FUNCTION_BLOCK FB_VRC_NO_FFO_VLS EXTENDS FB_VRC_NO
VAR_IN_OUT
    io_fbFFHWO    :    FB_HardwareFFOutput;
    fbArbiter: FB_Arbiter();
END_VAR
VAR_INPUT
    i_xPMPS_OK:	BOOL	; (*Set to True To switch off the bptm and PMPS Arbiter*)
    i_xIsAperture:BOOL :=FALSE; // Set tp True if this is an Aperture Valve, the MPS Fault will trip only when moving.
    i_sDevName : T_MaxString :=  'VGC'; // Device name for diagnostic
    i_nTransitionRootID: UDINT; //A unique transition Root ID that is equal to or greater than 1000i_xIsAperture:BOOL :=FALSE; // Set tp True if this is an Aperture Valve, the MPS Fault will trip only when moving.
END_VAR
VAR_OUTPUT

END_VAR
VAR

    xPMPS_OK:	BOOL	; (*PMPS interlock*)
    bMoving : BOOL;
    bDone :BOOL;
    tBPTMtimeout:TON;
    bptm: BeamParameterTransitionManager;
    FFO    :    FB_FastFault :=(
        i_DevName := 'VGC',
        i_Desc := 'Fault occurs when the valve is not in safe state',
        i_TypeCode := 16#1010);
    xMPS_OK:	BOOL; (*MPS Fast OK, is set when the Valve is Open*)

END_VAR

(*IO Mapping*)
ACT_IO();

(* On first PLC pass, put valve into vented state, which implies a closed valve *)
IF xFirstPass THEN
    iq_stValve.eVGC_State := Vented;
    iq_stValve.pv_xCLS_SW := FALSE;
    FFO.i_DevName := i_sDevName;
//	iq_stValve.sDevName := i_sDevName;
END_IF


///Check valve position
IF iq_stValve.i_xClsLS AND  iq_stValve.i_xOpnLS THEN
    iq_stValve.eState:=INVALID;
ELSIF NOT iq_stValve.i_xOpnLS AND iq_stValve.i_xClsLS AND iq_stValve. THEN
    iq_stValve.eState:=CLOSED;
ELSIF NOT iq_stValve.i_xClsLS AND iq_stValve.i_xOpnLS AND NOT iq_stValve.q_xOPN_DO THEN
    iq_stValve.eState:=OPEN_F;
ELSIF iq_stValve.i_xClsLS AND NOT iq_stValve.i_xOpnLS AND NOT iq_stValve.q_xOPN_DO THEN
    iq_stValve.eState:=CLOSED;
ELSIF NOT iq_stValve.i_xClsLS AND NOT iq_stValve.i_xOpnLS THEN
    iq_stValve.eState:=MOVING;
ELSE
    iq_stValve.eState:=INVALID;
END_IF




(*PMPS*)
IF NOT(i_xPMPS_OK) THEN
    ACT_PMPS();
END_IF
(*when interlock is lost the Valve closes regardless of the status of the PMPS and EPS*)
xPMPS_OK := i_xPMPS_OK OR (bptm.q_xTransitionAuthorized OR tBPTMtimeout.Q);
IF NOT (iq_stValve.xOPN_OK) THEN
    iq_stValve.pv_xOPN_SW:= FALSE; // Reset switch after inlk is lost
    iq_stValve.q_xOPN_DO := (iq_stValve.pv_xOPN_SW  AND iq_stValve.xOPN_OK) OR (tonOvrd.Q AND i_xOverrideMode);
ELSIF xPMPS_OK THEN
    iq_stValve.q_xOPN_DO := (iq_stValve.pv_xOPN_SW  AND iq_stValve.xOPN_OK) OR (tonOvrd.Q AND i_xOverrideMode);
//ELSIF NOT (i_xPMPS_OK) THEN
    // Only override mode
    //iq_stValve.q_xOPN_DO := (tonOvrd.Q AND i_xOverrideMode);
END_IF

(*MPS Fault setting*)
If (i_xIsAperture ) THEN
    (* When the valve  is open or in Closed position MPS is OK, Fault while moving*)
    xMPS_OK := (i_xOpnLS  AND NOT q_xCLS_DO) XOR (i_xClsLS  AND q_xCLS_DO);
ELSE
    (* When the valve  is open MPS is OK*)
    xMPS_OK := i_xOpnLS AND NOT i_xClsLS AND q_xCLS_DO;
END_IF

(*FAST FAULT*)
FFO(i_xOK := xMPS_OK,
    i_xReset := ,
    i_xAutoReset :=TRUE,
    io_fbFFHWO := io_fbFFHWO);

ACTION ACT_IO:
(*inputs*)
iq_stValve.i_xOpnLS := 	i_xOpnLS;
iq_stValve.i_xClsLS:=	i_xClsLS;
//iq_stValve. := i_xEXT_OK;
iq_stValve.xOverrideMode := i_xOverrideMode;
(*outputs*)
//q_xOPN_DO:= iq_stValve.q_xOPN_DO;
END_ACTION

ACTION ACT_PMPS:
bMoving := (iq_stValve.pv_xOPN_SW AND iq_stValve.i_xClsLS) XOR (NOT iq_stValve.pv_xOPN_SW AND i_xOpnLS);
bDone := (iq_stValve.pv_xOPN_SW AND iq_stValve.i_xOpnLS) XOR (NOT iq_stValve.pv_xOPN_SW AND i_xClsLS);
If (i_xIsAperture ) OR (iq_stValve.pv_xOPN_SW )THEN
    bptm.i_stRequestedAssertion := PMPS_GVL.cstFullBeam;
ELSE  bptm.i_stRequestedAssertion := PMPS_GVL.cst0RateBeam;
END_IF
bptm(fbArbiter:=fbArbiter,
     i_TransitionAssertionID:=i_nTransitionRootID+2,
     i_stTransitionAssertion:=PMPS_GVL.cst0RateBeam,
     i_nRequestedAssertionID:=i_nTransitionRootID+ BOOL_TO_UDINT( iq_stValve.pv_xOPN_SW),
     i_stRequestedAssertion:=,
     i_xMoving:=bMoving,
     i_xDoneMoving:= bDone,
     stCurrentBeamParameters:=PMPS_GVL.stCurrentBeamParameters,
     q_xTransitionAuthorized=>);
// Timeout
tBPTMtimeout(IN:= bMoving AND NOT bptm.q_xTransitionAuthorized , PT:=T#1S);
//xPMPS_OK := bptm.q_xTransitionAuthorized OR tBPTMtimeout.Q;

//Timeout and clear request
IF (tBPTMtimeout.Q) THEN
    fbArbiter.RemoveRequest(bptm.i_TransitionAssertionID);
    fbArbiter.RemoveRequest(bptm.i_nRequestedAssertionID);
END_IF
END_ACTION

METHOD PUBLIC M_IsClosed : BOOL
VAR_INPUT
END_VAR
M_IsClosed := (This^.iq_stValve.eState = E_ValvePositionState.CLOSED);
END_METHOD

METHOD PUBLIC M_IsOpen : BOOL
VAR_INPUT
END_VAR
M_IsOpen := (This^.iq_stValve.eState = E_ValvePositionState.OPEN);
END_METHOD

// Use this Methode to Open or close the valve by setting the OPN_SW to the input value.
METHOD PUBLIC M_Set_CLS_SW : BOOL
VAR_INPUT
        value:BOOL;
END_VAR
This^.iq_stValve.pv_xCLS_SW := value;
END_METHOD

END_FUNCTION_BLOCK

(* stored: Version 1.1.0.1, ProductVersion 3.1.4022.18
   POU FB_VRC_NO_FFO_VLS: Id {6c7b96aa-1e17-4f9d-82a3-e115363dfca4}, SpecialFunc None
   Action ACT_IO: Id {86d3dad0-9d99-4d69-8399-47f0b93aa886}
   Action ACT_PMPS: Id {1f5dca28-1929-4129-ad18-d7cc7c2735cf}
   Method M_IsClosed: Id {73d61226-05ce-4b07-b720-a4265f22b253}
   Method M_IsOpen: Id {6e28fe8a-152c-427f-915e-9ada086885d1}
   Method M_Set_CLS_SW: Id {f95a3e5e-d04c-419a-9bb5-06f554013cb0} *)
